// TIA Portal V20 export
TYPE "IO_Device_Conveyor_Belt_Ouput"
   STRUCT
      Start : Bool;
      Manual_Turn_On_Motor_Caroussel : Bool;
      Manual_Turn_On_Motor_Conveyor_Belt : Bool;
      Water_Foutain_Fail_Functional_Test : Bool;
      Select_Motor_Speed : SInt;
      Carousel_Voltage_Selection : SInt;
   END_STRUCT;
END_TYPE
